//{attribute 'qualified_only'}
VAR_GLOBAL
    //Fiber-Lite Control
    {attribute 'TcLinkTo' := '.iIlluminatorINT := TIID^Device 1 (EtherCAT)^Term 5 (EK1200)^Term 6 (EK1122-0080)^DRL02-EK0 (EK1101-0080)^DRL02-ECJ1 (EK1122)^CryoStat (EK1101)^Term 158 (EL4004)^AO Outputs Channel 1^Analog output'}
    {attribute 'pytmc' := '
        pv: RIX:CRIX:LED:01
        io: io
    '}

    bLedOutput1 : FB_LED;

    {attribute 'TcLinkTo' := '.iIlluminatorINT := TIID^Device 1 (EtherCAT)^Term 5 (EK1200)^Term 6 (EK1122-0080)^DRL02-EK0 (EK1101-0080)^DRL02-ECJ1 (EK1122)^CryoStat (EK1101)^FiberLite (EL4004)^AO Outputs Channel 2^Analog output'}
    {attribute 'pytmc' := '
        pv: RIX:CRIX:LED:02
        io: io
    '}

    bLedOutput2 : FB_LED;

       {attribute 'TcLinkTo' := '.iIlluminatorINT := TIID^Device 1 (EtherCAT)^Term 5 (EK1200)^Term 6 (EK1122-0080)^DRL02-EK0 (EK1101-0080)^DRL02-ECJ1 (EK1122)^CryoStat (EK1101)^FiberLite (EL4004)^AO Outputs Channel 3^Analog output'}
    {attribute 'pytmc' := '
        pv: RIX:CRIX:LED:03
        io: io
    '}

    bLedOutput3 : FB_LED;

       {attribute 'TcLinkTo' := '.iIlluminatorINT := TIID^Device 1 (EtherCAT)^Term 5 (EK1200)^Term 6 (EK1122-0080)^DRL02-EK0 (EK1101-0080)^DRL02-ECJ1 (EK1122)^CryoStat (EK1101)^FiberLite (EL4004)^AO Outputs Channel 4^Analog output'}
    {attribute 'pytmc' := '
        pv: RIX:CRIX:LED:04
        io: io
    '}

    bLedOutput4 : FB_LED;


    (*
    addding two digital outputs to be used for FZP-TXAS led control
    Beckhoff EL2004 FZP-TXAS-LED- 4 Digital Outputs
    Renamed variables to FZP_TXAS_LED_01–02
*)

     {attribute 'TcLinkTo' := 'TIID^Device 1 (EtherCAT)^Term 5 (EK1200)^Term 6 (EK1122-0080)^DRL02-EK0 (EK1101-0080)^DRL02-ECJ0 (EK1122-0080)^Term 109 (EK1101-0080)^FZP LED(EL2004)^Channel 1^Output'}
    {attribute 'pytmc' := '
        pv: RIX:CRIX:LED:05
        io: io
'}
FZP_TXAS_LED_01 AT %Q*:BOOL;


     {attribute 'TcLinkTo' :='TIID^Device 1 (EtherCAT)^Term 5 (EK1200)^Term 6 (EK1122-0080)^DRL02-EK0 (EK1101-0080)^DRL02-ECJ0 (EK1122-0080)^Term 109 (EK1101-0080)^FZP LED(EL2004)^Channel 2^Output'}
    {attribute 'pytmc' := '
        pv: RIX:CRIX:LED:06
        io: io
'}
FZP_TXAS_LED_02 AT %Q*: BOOL;

END_VAR

(* stored: Version 1.1.0.1, ProductVersion 3.1.4022.18
   GVL GVL_FiberLite: Id {226d6881-986f-4480-8f74-cd36d8198de3} *)
